FUNCTION_BLOCK E_TABLE_CTRL (* Support function block for E_TABLE *)
  (* Standard: 61499-1 Annex A; Description: Copyright (c) 2017 fortiss GmbH This program and the accompanying materials are made available under the terms of the Eclipse Public License 2.0 which is available at https://www.eclipse.org/legal/epl-2.0/ SPDX-License-Identifier: EPL-2.0 *)
  (* Version 1.0, 2017-09-22, Alois Zoitl, fortiss GmbH, initial API and implementation and/or initial documentation *)
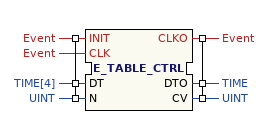
  EVENT_INPUT
    INIT WITH DT, N;
    CLK;
  END_EVENT
  EVENT_OUTPUT
    CLKO WITH DTO, CV;
  END_EVENT
  VAR_INPUT
    DT : ARRAY [0..3] OF TIME;
    N : UINT;
  END_VAR
  VAR_OUTPUT
    DTO : TIME;
    CV : UINT;
  END_VAR
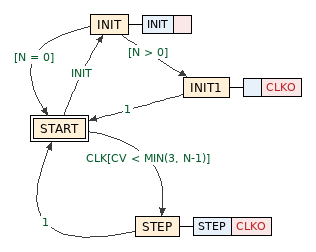
  EC_STATES
    START; (* Initial State *)
    INIT : INIT;
    INIT1 : -> CLKO;
    STEP : STEP -> CLKO;
  END_STATES
  EC_TRANSITIONS
    START TO INIT := INIT;
    INIT TO START := [N = 0];
    INIT TO INIT1 := [N > 0];
    INIT1 TO START := 1;
    START TO STEP := CLK[CV < MIN(3, N-1)];
    STEP TO START := 1;
  END_TRANSITIONS
  ALGORITHM INIT IN ST: (* new algorithm *)
CV := 0;
DTO := DT[0];
  END_ALGORITHM
  ALGORITHM STEP IN ST: (* new algorithm *)
CV := CV +1;
DTO := DT[CV];
  END_ALGORITHM
END_FUNCTION_BLOCK
